// TIA Portal V20 export
TYPE "LER_typeCommunicationDataI2S"
// stored: Access Published
   STRUCT
      UnitStatus : "LER_typeCommunicationUnitStatus";
      UnitHmiData : Array[1..50] of "LER_typeUnitHmiData";
      InterfaceData : "LER_typeCommunicationInterfaceData";
   END_STRUCT;
END_TYPE
